// Mitsubishi GX Works2 project: z19   PLC: Q02/Q02H

PROGRAM MAIN
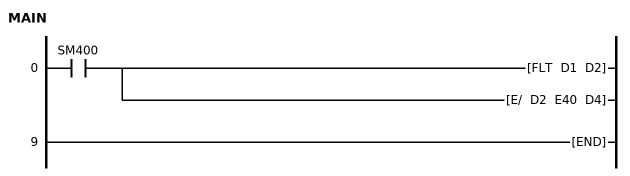
0     LD      SM400
      FLT     D1 D2
      E/      D2 E40 D4
9     END
END_PROGRAM
